(* CODESYS project testModbus.project

Project tree, tasks and I/O mapping:
  Device : Jinan Cherry-ARM Cortex-VxWorks, Jinan Cheery Electric Co., Ltd., version 3.5.11.20
    application Application
      libraries: Standard, * (System); File Access, 3.5.7.0 (3S - Smart Software Solutions GmbH); CmpModbusLib, 1.0.0 (HiTech)
      task MainTask (cyclic, interval 500 ms, priority 1) calls PLC_PRG
      program PLC_PRG [ST]
    SoftMotion General Axis Pool
*)

// Device/Application/PLC_PRG
PROGRAM PLC_PRG
VAR
	initModbus : CmpModbusLib.InitModbusRtu;
	readReg	   : CmpModbusLib.ModbusReadReg;
	writeReg   : CmpModbusLib.ModbusWriteReg;
	readBit    : CmpModbusLib.ModbusReadBit;
	writeBit   : CmpModbusLib.ModbusWriteBit;
	readSlaveBit  : CmpModbusLib.ModbusSlaveReadBit;
	writeSlaveBit : CmpModbusLib.ModbusSlaveWriteBit;
	fileOpen : FILE.Open;
	//flag value
	initOK : BOOL := FALSE;
	result : INT;
	i:INT;
	
	//Comm Data
	regWord : ARRAY[0..31] OF WORD;	
	regByte : ARRAY[0..31] OF BYTE;
	slaveBitData : ARRAY[0..255] OF USINT;	
	slaveRegData : ARRAY[0..255] OF UINT;	
	//Screen Data
	start : BOOL;
	number : WORD := 0;
	data : ARRAY[0..3] OF WORD;
	slaveData : USINT;
	
	//IO Data
	button : BOOL;
	led : BOOL;
END_VAR
VAR_INPUT
END_VAR
VAR_IN_OUT
END_VAR

IF initOK = FALSE THEN
	initModbus(
		com:= 3, 
		baud:= 9600,
		slave:= 1, 
		timeout:= 100, 
		result=> result);
	IF result = 0 THEN
		initOK := TRUE;
	END_IF
ELSE
	//根数
	//readReg(addr := 1, num := 1, data := regWord);
	//number := regWord[0];	
	
	//钢筋数据
	//readReg(addr := 10, num := 4, data := regWord);	
	//FOR i := 0 TO 3 BY +1 DO
	//	data[i] := regWord[i];		
	//END_FOR
	
	//开始
	//readBit(addr := 0, num := 1, data := regByte);
	//start := BYTE_TO_BOOL(regByte[0]);
	
	//readSlaveBit(addr := 0, num := 4, data := slaveBitData);
	button := NOT button;
	slaveBitData[0] := BOOL_TO_USINT(button);
	writeSlaveBit(addr := 0, num := 4, data := slaveBitData);
END_IF

END_PROGRAM
